(* IEC 61131-3 sources: Industry-PLC-LLM/data/PLCBEAD_repo/PLCBEAD_PLCEmbed-main/PLC-BEAD/Source/GEB/TANC, 1 file *)

(* ---- TANC.ST ---- *)
FUNCTION TANC:REAL

	VAR_INPUT
		X :	REAL;
	END_VAR

	IF X = 0.0 THEN
		TANC := 1.0;
	ELSE
		TANC := TAN(X) / x;
	END_IF;

END_FUNCTION

PROGRAM program0

	VAR
		X :	REAL;
		CEIL5_OUT : REAL;
	END_VAR

	CEIL5_OUT := TANC(X);

END_PROGRAM
